# EPICS substitutions: BoxStatusTestApp/Db/test.substitutions
# $File: //ASP/tec/epics/boxStatus/trunk/BoxStatusTestApp/Db/test.substitutions $
# $Revision: #2 $
# $DateTime: 2023/05/13 14:49:10 $
# Last checked in by: $Author: starritt $
#

file db/Box_Status.template {
   pattern { BOX,               FUNCTION,    LOCATION  }
           { "K01",             "",          ""        }
           { "K02",             "",          ""        }
           { "K03",             "",          ""        }
           { "K04",             "",          ""        }
           { "K05",             "",          ""        }
           { "K06",             "",          ""        }
           { "K07",             "",          ""        }
           { "K08",             "",          ""        }
           { "K09",             "",          ""        }
           { "K10",             "",          ""        }
           { "K11",             "",          ""        }
           { "K12",             "",          ""        }
           { "K13",             "",          ""        }
           { "K14",             "",          ""        }
           { "K15",             "",          ""        }
           { "K16",             "",          ""        }
           { "K17",             "",          ""        }
           { "K18",             "",          ""        }
           { "K19",             "",          ""        }
           { "K20",             "",          ""        }
           { "K21",             "",          ""        }
           { "K22",             "",          ""        }
           { "K23",             "",          ""        }
           { "K24",             "",          ""        }
           { "K25",             "",          ""        }
           { "K26",             "",          ""        }
           { "K27",             "",          ""        }
           { "K28",             "",          ""        }
           { "K29",             "",          ""        }
           { "K30",             "",          ""        }
}

# end
